% RSLogix 500 project I2P-JOB-10 DUNCAN_SUTTON.RSS, saved by version 10.00.00.00 %
PROJECT "ML01A"    % processor: Bul.1763 MicroLogix 1100 Series B %

PROGRAM FILES
  LAD 2   6 rungs

DATA FILES
  O0 OUTPUT  4 elements
  I1 INPUT  6 elements
  S2 STATUS  66 elements
  B3 BINARY  1 elements
  T4 TIMER  1 elements
  C5 COUNTER  1 elements
  R6 CONTROL  1 elements
  N7 INTEGER  1 elements
  F8 FLOAT  1 elements

LADDER 2
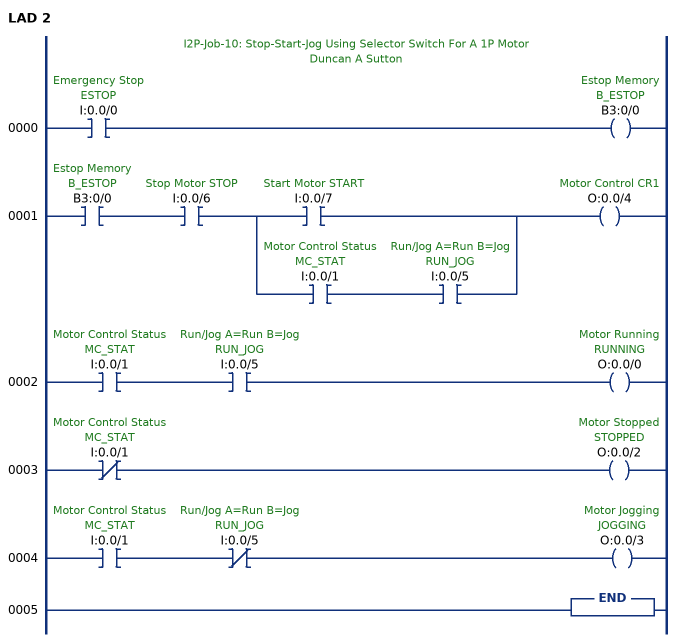
% Rung: 0 %
% I2P-Job-10: Stop-Start-Jog Using Selector Switch For A 1P Motor
% Duncan A Sutton %
SOR XIC I:0.0/0 OTE B3:0/0 EOR
%   I:0.0/0  ESTOP  "Emergency Stop" %
%   B3:0/0  B_ESTOP  "Estop Memory" %
% Rung: 1 %
SOR XIC B3:0/0 XIC I:0.0/6 BST XIC I:0.0/7 NXB XIC I:0.0/1 XIC I:0.0/5 BND OTE O:0.0/4 EOR
%   B3:0/0  B_ESTOP  "Estop Memory" %
%   I:0.0/6  STOP  "Stop Motor" %
%   I:0.0/7  START  "Start Motor" %
%   I:0.0/1  MC_STAT  "Motor Control Status" %
%   I:0.0/5  RUN_JOG  "Run/Jog A=Run B=Jog" %
%   O:0.0/4  CR1  "Motor Control" %
% Rung: 2 %
SOR XIC I:0.0/1 XIC I:0.0/5 OTE O:0.0/0 EOR
%   I:0.0/1  MC_STAT  "Motor Control Status" %
%   I:0.0/5  RUN_JOG  "Run/Jog A=Run B=Jog" %
%   O:0.0/0  RUNNING  "Motor Running" %
% Rung: 3 %
SOR XIO I:0.0/1 OTE O:0.0/2 EOR
%   I:0.0/1  MC_STAT  "Motor Control Status" %
%   O:0.0/2  STOPPED  "Motor Stopped" %
% Rung: 4 %
SOR XIC I:0.0/1 XIO I:0.0/5 OTE O:0.0/3 EOR
%   I:0.0/1  MC_STAT  "Motor Control Status" %
%   I:0.0/5  RUN_JOG  "Run/Jog A=Run B=Jog" %
%   O:0.0/3  JOGGING  "Motor Jogging" %
% Rung: 5 %
SOR END EOR

OTHER DOCUMENTED ADDRESSES
  I:0.0/2  CR2_C  "Control Relay 2 Contact"
  I:0.0/3  3PSS_PA  "3 Postion Selector Switch Position A"
  I:0.0/4  3PSS_PB  "3 Position Selector Switch Position B"
  I:0.0/8  PB_3  "Pushbutton 3"
  O:0.0/1  "Yellow Light"
  O:0.0/5  CR_2  "Control Relay 2"

DATA TABLE (non-zero values as saved)
DATA B3
% B3:0 % 0X0001
